PROGRAM SFCMotor
VAR
	PushPopFB_0: PushPopFB;
	TargFloor: UINT;
	OutputFloor: UINT;
	MemoryMotor: UINT;

END_VAR
VAR // added by the converter: edge detectors and wires of the graphical bodies
    _rt1, _rt2, _rt3 : R_TRIG;
    _w1, _w2, _w3 : BOOL;
END_VAR

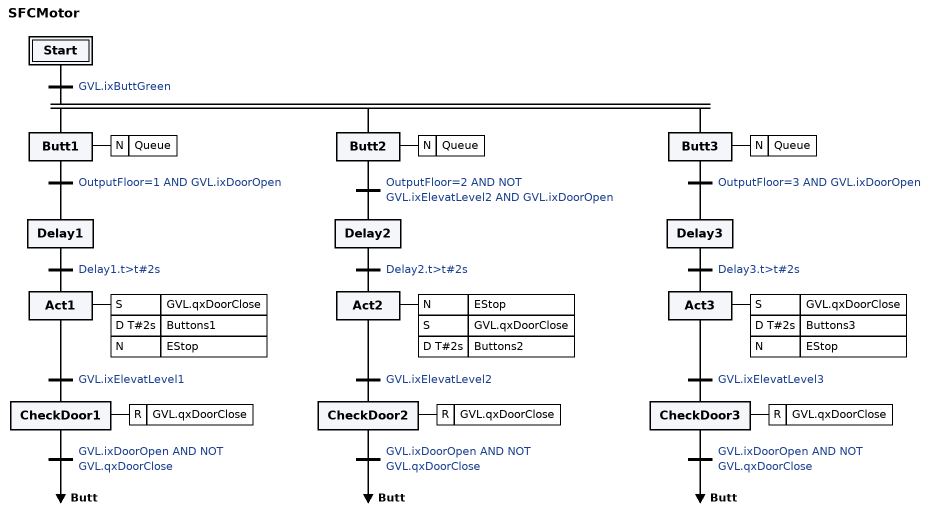
INITIAL_STEP Start:
END_STEP
TRANSITION FROM Start TO (Butt1, Butt2, Butt3)
    := GVL.ixButtGreen;
END_TRANSITION
STEP Butt1:
    Queue(N);
END_STEP
STEP Butt2:
    Queue(N);
END_STEP
TRANSITION FROM Butt2 TO Delay2
    := OutputFloor=2 AND NOT GVL.ixElevatLevel2 AND GVL.ixDoorOpen;
END_TRANSITION
STEP Delay2:
END_STEP
TRANSITION FROM Delay2 TO Act2
    := Delay2.t>t#2s;
END_TRANSITION
STEP Act2:
    EStop(N);
    GVL.qxDoorClose(S);
    Buttons2(D, T#2s);
END_STEP
TRANSITION FROM Act2 TO CheckDoor2
    := GVL.ixElevatLevel2;
END_TRANSITION
STEP CheckDoor2:
    GVL.qxDoorClose(R);
END_STEP
TRANSITION FROM CheckDoor2 TO (Butt1, Butt2, Butt3)
    := GVL.ixDoorOpen AND NOT GVL.qxDoorClose;
END_TRANSITION
STEP Butt3:
    Queue(N);
END_STEP
TRANSITION FROM Butt3 TO Delay3
    := OutputFloor=3 AND GVL.ixDoorOpen;
END_TRANSITION
STEP Delay3:
END_STEP
TRANSITION FROM Delay3 TO Act3
    := Delay3.t>t#2s;
END_TRANSITION
STEP Act3:
    GVL.qxDoorClose(S);
    Buttons3(D, T#2s);
    EStop(N);
END_STEP
TRANSITION FROM Act3 TO CheckDoor3
    := GVL.ixElevatLevel3;
END_TRANSITION
STEP CheckDoor3:
    GVL.qxDoorClose(R);
END_STEP
TRANSITION FROM CheckDoor3 TO (Butt1, Butt2, Butt3)
    := GVL.ixDoorOpen AND NOT GVL.qxDoorClose;
END_TRANSITION
TRANSITION FROM Butt1 TO Delay1
    := OutputFloor=1 AND GVL.ixDoorOpen;
END_TRANSITION
STEP Delay1:
END_STEP
TRANSITION FROM Delay1 TO Act1
    := Delay1.t>t#2s;
END_TRANSITION
STEP Act1:
    GVL.qxDoorClose(S);
    Buttons1(D, T#2s);
    EStop(N);
END_STEP
TRANSITION FROM Act1 TO CheckDoor1
    := GVL.ixElevatLevel1;
END_TRANSITION
STEP CheckDoor1:
    GVL.qxDoorClose(R);
END_STEP
TRANSITION FROM CheckDoor1 TO (Butt1, Butt2, Butt3)
    := GVL.ixDoorOpen AND NOT GVL.qxDoorClose;
END_TRANSITION
// branch label Butt

ACTION Buttons1:

IF GVL.ixDoorClosed THEN
	
	IF GVL.ixElevatLevel2 OR GVL.ixElevatLevel3 THEN
		GVL.qxMotorDown := TRUE;
	END_IF

	IF GVL.ixElevatLevel1  THEN
		GVL.qxMotorDown :=FALSE;
		GVL.qxMotorUp :=FALSE;
	END_IF
END_IF
END_ACTION

ACTION Buttons2:
IF GVL.ixDoorClosed THEN
	IF GVL.ixElevatLevel1 THEN
		GVL.qxMotorUp := TRUE;
	END_IF

	IF GVL.ixElevatLevel3  THEN
		GVL.qxMotorDown :=TRUE;
	END_IF

	IF GVL.ixElevatLevel2  THEN
		GVL.qxMotorDown :=FALSE;
		GVL.qxMotorUp :=FALSE;
	END_IF
END_IF
END_ACTION

ACTION Buttons3:
IF GVL.ixDoorClosed THEN
	
	IF GVL.ixElevatLevel2 OR GVL.ixElevatLevel1 THEN
		GVL.qxMotorUp := TRUE;
	END_IF

	IF GVL.ixElevatLevel3  THEN
		GVL.qxMotorDown :=FALSE;
		GVL.qxMotorUp :=FALSE;
	END_IF
END_IF
END_ACTION

ACTION CheckDoor:


IF GVL.ixDoorClosed THEN
	GVL.qxDoorClose := FALSE;
END_IF
END_ACTION

ACTION EStop:


IF NOT GVL.ixButtRed  THEN
	IF GVL.qxMotorDown THEN
		GVL.qxMotorDown :=FALSE;
		MemoryMotor :=2;
	
	ELSIF GVL.qxMotorUp THEN
		GVL.qxMotorUp :=FALSE;
		MemoryMotor :=1;
	
	END_IF
END_IF

IF GVL.ixButtGreen AND MemoryMotor>0 THEN
	IF OutputFloor=2 AND MemoryMotor=1 THEN
		GVL.qxMotorUp:=TRUE;
		MemoryMotor:=0;
	END_IF

	IF OutputFloor=2 AND MemoryMotor=2 THEN
		GVL.qxMotorDown:=TRUE;
		MemoryMotor:=0;
	END_IF

	IF OutputFloor=1 AND MemoryMotor=2 THEN
		GVL.qxMotorDown:=TRUE;
		MemoryMotor:=0;
	END_IF

	IF OutputFloor=3 AND MemoryMotor=1 THEN
		GVL.qxMotorUp:=TRUE;
		MemoryMotor:=0;
	END_IF
END_IF
END_ACTION

ACTION Queue:
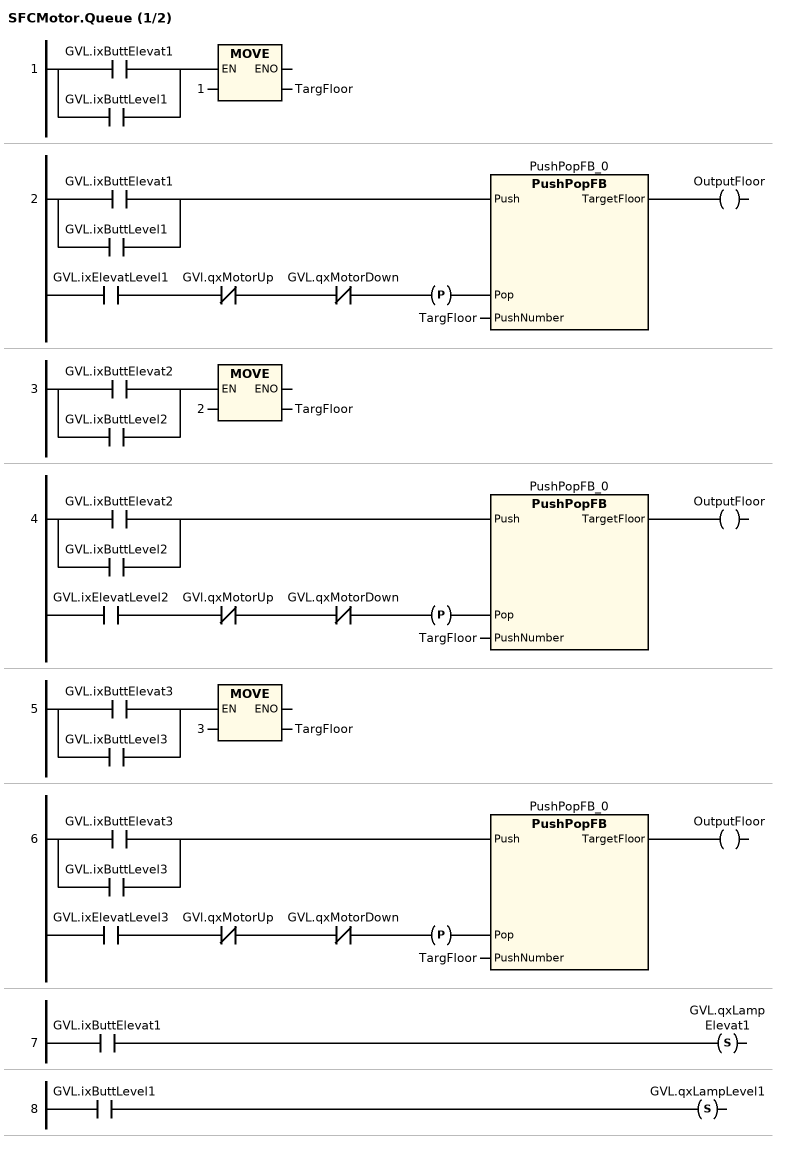
// NETWORK 1
IF GVL.ixButtElevat1 OR GVL.ixButtLevel1 THEN TargFloor := 1; END_IF

// NETWORK 2
_rt1(CLK := GVL.ixElevatLevel1 AND NOT GVl.qxMotorUp AND NOT GVL.qxMotorDown);
PushPopFB_0(Push := GVL.ixButtElevat1 OR GVL.ixButtLevel1, Pop := _rt1.Q, PushNumber := TargFloor); // PushPopFB
OutputFloor := PushPopFB_0.TargetFloor;

// NETWORK 3
IF GVL.ixButtElevat2 OR GVL.ixButtLevel2 THEN TargFloor := 2; END_IF

// NETWORK 4
_rt2(CLK := GVL.ixElevatLevel2 AND NOT GVl.qxMotorUp AND NOT GVL.qxMotorDown);
PushPopFB_0(Push := GVL.ixButtElevat2 OR GVL.ixButtLevel2, Pop := _rt2.Q, PushNumber := TargFloor); // PushPopFB
OutputFloor := PushPopFB_0.TargetFloor;

// NETWORK 5
IF GVL.ixButtElevat3 OR GVL.ixButtLevel3 THEN TargFloor := 3; END_IF

// NETWORK 6
_rt3(CLK := GVL.ixElevatLevel3 AND NOT GVl.qxMotorUp AND NOT GVL.qxMotorDown);
PushPopFB_0(Push := GVL.ixButtElevat3 OR GVL.ixButtLevel3, Pop := _rt3.Q, PushNumber := TargFloor); // PushPopFB
OutputFloor := PushPopFB_0.TargetFloor;

// NETWORK 7
GVL.qxLampElevat1 S= GVL.ixButtElevat1;

// NETWORK 8
GVL.qxLampLevel1 S= GVL.ixButtLevel1;

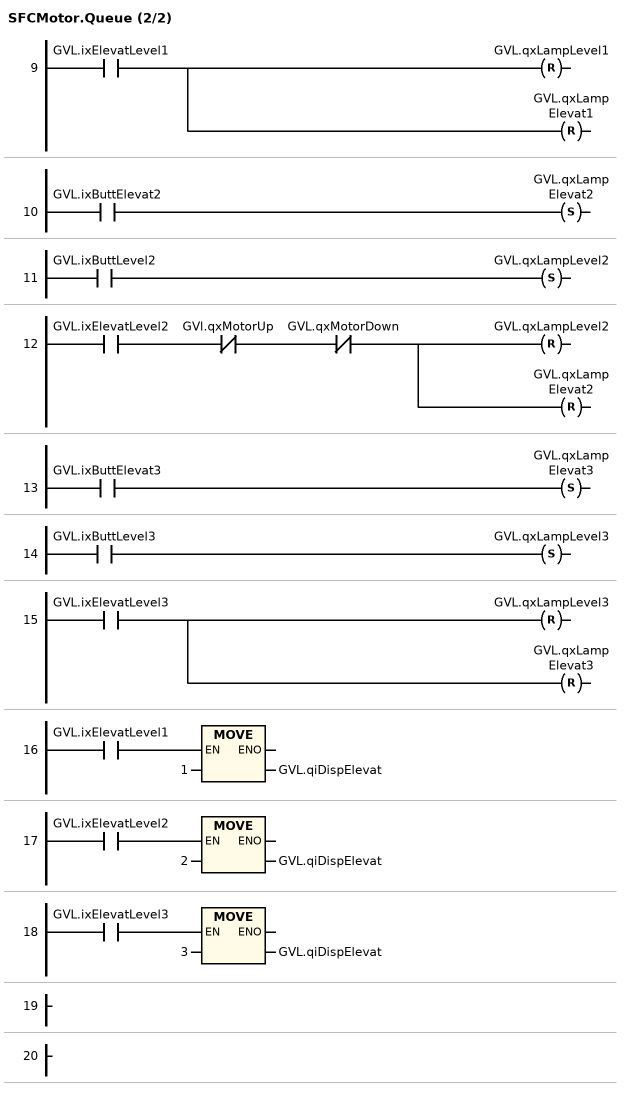
// NETWORK 9
_w1 := GVL.ixElevatLevel1;
GVL.qxLampLevel1 R= _w1;
GVL.qxLampElevat1 R= _w1;

// NETWORK 10
GVL.qxLampElevat2 S= GVL.ixButtElevat2;

// NETWORK 11
GVL.qxLampLevel2 S= GVL.ixButtLevel2;

// NETWORK 12
_w2 := GVL.ixElevatLevel2 AND NOT GVl.qxMotorUp AND NOT GVL.qxMotorDown;
GVL.qxLampLevel2 R= _w2;
GVL.qxLampElevat2 R= _w2;

// NETWORK 13
GVL.qxLampElevat3 S= GVL.ixButtElevat3;

// NETWORK 14
GVL.qxLampLevel3 S= GVL.ixButtLevel3;

// NETWORK 15
_w3 := GVL.ixElevatLevel3;
GVL.qxLampLevel3 R= _w3;
GVL.qxLampElevat3 R= _w3;

// NETWORK 16
IF GVL.ixElevatLevel1 THEN GVL.qiDispElevat := 1; END_IF

// NETWORK 17
IF GVL.ixElevatLevel2 THEN GVL.qiDispElevat := 2; END_IF

// NETWORK 18
IF GVL.ixElevatLevel3 THEN GVL.qiDispElevat := 3; END_IF

// NETWORK 19

// NETWORK 20
END_ACTION

END_PROGRAM

(* stored: Version 1.1.0.1, ProductVersion 3.1.4024.12
   POU SFCMotor: Id {b1d49eca-8be5-4bb5-a036-e2e39d4e04b2}, SpecialFunc None
   Action Buttons1: Id {6a1b36c3-5e15-4cbb-8fd1-5ee1f79ec100}
   Action Buttons2: Id {93961a2b-749c-4007-8a8d-939ba09610de}
   Action Buttons3: Id {2d5ae051-27ca-4d80-a968-7c11806f832b}
   Action CheckDoor: Id {bb4829d4-d298-41f1-a7a1-c246ee1048cc}
   Action EStop: Id {844dc8f9-b87c-4d7f-8d16-6804d254ab86}
   Action Queue: Id {ec19e23a-1931-4484-ba83-5fe553fd6c6a} *)
